FUNCTION_BLOCK ManipulateFunctionsTest EXTENDS TcUnit.FB_TestSuite
VAR
END_VAR

AddLeadingZerosFunction();
GetStringBetweenFunction();
RemoveStringFromEndFunction();
ReplaceStringFunction();
ReplaceAllFunction();
ReplaceAllAnyFunction();
ReplaceAllAnyTypeFunction();
SubstringFunction();

METHOD AddLeadingZerosFunction : BOOL
VAR
	test : T_MaxString := '555';
END_VAR
TcUnit.TEST('Add leading zeros');

AssertEquals_STRING(
	Expected := '00555',
	Actual := AddLeadingZeros(test, 5),
	Message := 'Should pad propper number of zeros');

AssertEquals_STRING(
	Expected := '555',
	Actual := AddLeadingZeros(test, 2),
	Message := 'Should do nothing if formatter string already has more chars');

TEST_FINISHED();
END_METHOD

METHOD GetStringBetweenFunction : BOOL
VAR
	test0 : T_MaxString := '1';
	test1 : T_MaxString := '[2]';
	test2 : T_MaxString := 'TestValue[3]rest';
	actual : T_MaxString;
END_VAR
TcUnit.TEST('Get string between');

actual := GetStringBetween(test0, '[', ']');

AssertEquals_STRING(
	Expected := '',
	Actual := actual,
	Message := 'Should return nothing');

actual := GetStringBetween(test1, '[', ']');

AssertEquals_STRING(
	Expected := '2',
	Actual := actual,
	Message := 'Should return content of brackets');

actual := GetStringBetween(test2, '[', ']');

AssertEquals_STRING(
	Expected := '3',
	Actual := actual,
	Message := 'Should return content of brackets');

TEST_FINISHED();
END_METHOD

METHOD RemoveStringFromEndFunction : BOOL
VAR
	test : T_MaxString := 'Last word will be removed';
	actual : T_MaxString;
END_VAR
TcUnit.TEST('Remove string from end');

actual := RemoveStringFromEnd(test, 'removed');

AssertEquals_STRING(
	Expected := 'Last word will be ',
	Actual := actual,
	Message := 'Should remove last word from test string');

TEST_FINISHED();
END_METHOD

METHOD ReplaceAllAnyFunction
VAR  
	inputString : T_MaxString;
	substringToReplace : T_MaxString;
	replacementSubstring : T_MaxString;
	inputAny, expectedAny : __SYSTEM.AnyType;
END_VAR
TcUnit.TEST('ReplaceAllAny Replaces Target Substring Correctly');
 
inputString  := 'Valve1 is open'; 
substringToReplace := 'Valve1';
replacementSubstring  := 'Valve2';
inputAny.diSize := SIZEOF(inputString);
inputAny.pValue := ADR(inputString); 
StringToAny('Valve2 is open',expectedAny);

ReplaceAllAny(inputAny,substringToReplace,replacementSubstring); 

AssertEquals_STRING(
	Expected := AnyToString(expectedAny),
	Actual := AnyToString(inputAny),
	Message := 'Should delete the substring if replacement is empty');

TEST_FINISHED();

//TcUnit.TEST('ReplaceAllAny Replaces Target Substring Correctly');
 
//inputString := 'Valve1 is open'; 
//substringToReplace := 'Valve1';
//replacementSubstring := 'Valve2';
//_toAnyType := ToAnyType(inputString);
//inputAny.diSize := SIZEOF(inputString);
//inputAny.pValue := ADR(inputString);

//ReplaceAllAny(inputAny,substringToReplace,replacementSubstring); 

//AssertEquals_STRING(
//	Expected := 'Valve2 is open',
//	Actual   := inputString,
//	Message  := 'Should delete the substring if replacement is empty');

//TEST_FINISHED();
END_METHOD

METHOD ReplaceAllAnyTypeFunction
VAR  
	inputString  : T_MaxString;
	_toAnyType : __SYSTEM.AnyType;
	substringToReplace : T_MaxString;
	replacementSubstring : T_MaxString;
END_VAR
TcUnit.TEST('ReplaceAllAnyType Replaces Target Substring Correctly');
 
inputString  := 'Valve1 is open'; 
substringToReplace := 'Valve1';
replacementSubstring  := 'Valve2';
_toAnyType := ToAnyType(inputString);

ReplaceAllAnyType(_toAnyType,substringToReplace,replacementSubstring); 

AssertEquals_STRING(
	Expected := 'Valve2 is open',
	Actual := AnyTypeToString(_toAnyType),
	Message := 'Should delete the substring if replacement is empty');

TEST_FINISHED();
END_METHOD

METHOD ReplaceAllFunction
VAR
	inputString  : T_MaxString;
	substringToReplace : T_MaxString;
	replacementSubstring  : T_MaxString;
END_VAR
TcUnit.TEST('ReplaceAll Replaces Target Substring Correctly');

inputString  := 'Valve1 is open';
substringToReplace := 'Valve1';
replacementSubstring  := 'Valve2';
 

AssertEquals_STRING(
	Expected := 'Valve2 is open',
	Actual := ReplaceAll(inputString,substringToReplace,replacementSubstring),
	Message := 'ReplaceAll should correctly replace the target substring in the input string');
	
inputString  := 'Valve1 is open';
substringToReplace := 'Valve4';
replacementSubstring  := 'Valve2';

AssertEquals_STRING(
	Expected := 'Valve1 is open',
	Actual := ReplaceAll(inputString,substringToReplace,replacementSubstring),
	Message := 'Should not modify the string if no match is found');
	
inputString  := 'Valve1 is open';
substringToReplace := 'Valve1';
replacementSubstring  := '';

AssertEquals_STRING(
	Expected := ' is open',
	Actual := ReplaceAll(inputString,substringToReplace,replacementSubstring),
	Message := 'Should delete the substring if replacement is empty');

TEST_FINISHED();
END_METHOD

METHOD ReplaceStringFunction : BOOL
VAR
	test : T_MaxString := 'this is test string';
END_VAR
TcUnit.TEST('Replace string');

ReplaceString(test, 'not here', 'replaced');

AssertEquals_STRING(
	Expected := 'this is test string',
	Actual := test,
	Message := 'Should do nothing because searched string is not there');

ReplaceString(test, 'test', 'replaced');

AssertEquals_STRING(
	Expected := 'this is replaced string',
	Actual := test,
	Message := 'Should replace found string');

TEST_FINISHED();
END_METHOD

METHOD SubstringFunction
VAR
	source : T_MaxString :=  'ABCDEF123456789';
	destination : T_MaxString;
	anySource : __SYSTEM.AnyType;
    anyDest : __SYSTEM.AnyType;
	startIndex : DINT := 3; 
    length : DINT := 5;
END_VAR
TcUnit.TEST('SubString Test');


anySource.pValue := ADR(source);
anySource.diSize := SIZEOF(source);
	
anyDest.pValue := ADR(destination);
anyDest.diSize := SIZEOF(destination);
	
SubString(source,destination,startIndex,length);
destination[LEN(destination)] := TO_BYTE(0);

//------------------EXP: DEF12, ACT: DEF12¨ÿÿ°----------------------

AssertEquals_STRING(Expected := 'DEF12',
					Actual :=  destination, 
					Message := 'Substring result incorrect');

TEST_FINISHED();
END_METHOD

END_FUNCTION_BLOCK

(* stored: Version 1.1.0.1, ProductVersion 3.1.4024.12
   POU ManipulateFunctionsTest: Id {8e2fe8b8-5e6f-0d30-1f80-87f977530bb8}, SpecialFunc None
   Method AddLeadingZerosFunction: Id {5b38fdb2-8f15-0071-0faa-54d830637f22}
   Method GetStringBetweenFunction: Id {adc4369a-6eeb-0f97-0df0-a2d6e56b181f}
   Method RemoveStringFromEndFunction: Id {3772e17f-2221-0625-2684-3b1eb052ea32}
   Method ReplaceAllAnyFunction: Id {b0638fe4-fb86-0b5b-2035-c1a68e913d99}
   Method ReplaceAllAnyTypeFunction: Id {89eacb8d-99ad-053a-0232-ab4ea4fe81d2}
   Method ReplaceAllFunction: Id {5c618a13-ecfa-0a46-0059-a8989e9615de}
   Method ReplaceStringFunction: Id {1ccb17b8-aa17-00ee-1667-3fe3bf06c9ae}
   Method SubstringFunction: Id {ca36775e-eb93-0de9-16dc-c9e64461a584} *)
